// TIA Portal V18 export
DATA_BLOCK "05_EM_STATE"   // DB7, F_DB
{ S7_Optimized_Access := 'TRUE'; DB_Accessible_From_OPC_UA := 'FALSE' }
VERSION : 0.1
// stored: AutoNumber true, DBAccessibleFromOPCUA false, DBAccessibleFromWebserver true
   VAR
      "AREA 1 Q" : Bool;   // Per-area emergency state (referenced by the 04/05/08 builders)
      "AREA 2 Q" : Bool;   // Per-area emergency state (referenced by the 04/05/08 builders)
      "AREA 3 Q" : Bool;   // Per-area emergency state (referenced by the 04/05/08 builders)
      "AREA 4 Q" : Bool;   // Per-area emergency state (referenced by the 04/05/08 builders)
      "AREA 1 Q_Delayed" : Bool;
      "AREA 2 Q_Delayed" : Bool;
      "AREA 3 Q_Delayed" : Bool;
      "AREA 4 Q_Delayed" : Bool;
      "AREA 1 RESET" : Bool;
      "AREA 2 RESET" : Bool;
      "AREA 3 RESET" : Bool;
      "AREA 4 RESET" : Bool;
      "AREA 1 POWER_CUT" : Bool;   // Per-area emergency power-cut coil written by the 04_ESTOP block (v1.1: one per area - was the sorter-only literal AREA 1 POWER_CUT; the _SAFETY_BREAKERS_COM/_SAFETY_DOORS_COM intermediates moved to the 02_COM cumulatives)
      "AREA 2 POWER_CUT" : Bool;   // Per-area emergency power-cut coil written by the 04_ESTOP block (v1.1: one per area - was the sorter-only literal AREA 1 POWER_CUT; the _SAFETY_BREAKERS_COM/_SAFETY_DOORS_COM intermediates moved to the 02_COM cumulatives)
      "AREA 3 POWER_CUT" : Bool;   // Per-area emergency power-cut coil written by the 04_ESTOP block (v1.1: one per area - was the sorter-only literal AREA 1 POWER_CUT; the _SAFETY_BREAKERS_COM/_SAFETY_DOORS_COM intermediates moved to the 02_COM cumulatives)
      "AREA 4 POWER_CUT" : Bool;   // Per-area emergency power-cut coil written by the 04_ESTOP block (v1.1: one per area - was the sorter-only literal AREA 1 POWER_CUT; the _SAFETY_BREAKERS_COM/_SAFETY_DOORS_COM intermediates moved to the 02_COM cumulatives)
      SORTER_01_NOT_RUNNING : Bool;   // One per sorter - nn = the safety-encoder index (as builders 07/08 number the sorters)
      SORTER_02_NOT_RUNNING : Bool;   // One per sorter - nn = the safety-encoder index (as builders 07/08 number the sorters)
   END_VAR
BEGIN
END_DATA_BLOCK
